Universal Robots PolyScope program: prac1_sergiorodriguez.urp

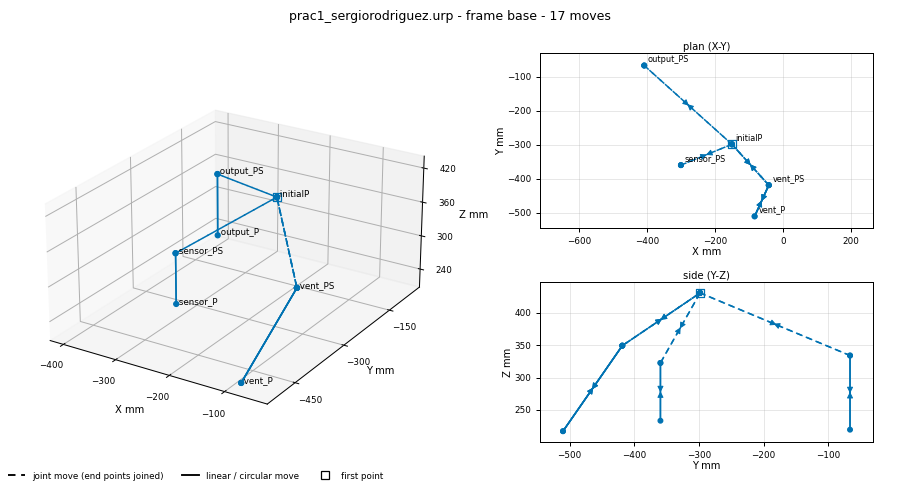
[picture p0: tool path of prac1_sergiorodriguez.urp in frame base, 17 of 17 moves have a stored position in this frame; points joined in program order, loops and branches not executed]
Program prac1_sergiorodriguez (installation=default directory=/programs createdIn=5.9.3.1031212 lastSavedIn=5.9.3.1031212 robotSerialNumber=20195300809)
Calibrated DH parameters: a=[-0.000085, -0.20076, -0.212369, 0.000121, -0.000118, 0]; d=[0.15185, -26.306375, 24.753047, 1.684739, 0.085386, 0.092088]; alpha=[1.572149, -0.00522, -0.011864, 1.571339, -1.571085, 0]; deltaTheta=[0, 0.599885, -0.513355, -0.086555, 0.000006, 0]
Robot Program (runOnlyOnce=false)
  URCap Gripper Activate (Robotiq_Grippers, Robotiq Inc.) dataModel(ResetAndActivateKey=false)
  URCap Gripper (Robotiq_Grippers, Robotiq Inc.) dataModel(position=0.0, force=100.0, speed=100.0, positionInDouble=0.0, forceInDouble=100.0, speedInDouble=100.0, slaveIds=[9], blocking=true)
  MoveJ speed 60 deg/s, acceleration 80 deg/s^2 (useActiveTCP=true) feature=Base
    Waypoint initialP: TCP in base x=-150.366 y=-298.238 z=430.772 mm, rx=1.2434 ry=2.8802 rz=0.0051 rad; joints [39.84, -76.565, 37.853, 308.981, -90.564, -2.908] deg
  Wait DigitalInput pin=digital_in[0]; digitalValue=1
  Wait Sleep waitTime=2.5
  MoveJ speed 60 deg/s, acceleration 80 deg/s^2 (useActiveTCP=true) feature=Base
    Waypoint sensor_PS: TCP in base x=-300.616 y=-359.588 z=322.64 mm, rx=0.0335 ry=-3.1211 rz=-0.1077 rad; joints [34.606, -41.931, 13.866, 299.406, -94.705, -56.283] deg
  MoveL speed 250 mm/s, acceleration 1200 mm/s^2 (useActiveTCP=true) feature=Base
    Waypoint sensor_P: TCP in base x=-300.596 y=-359.606 z=233.321 mm, rx=0.0335 ry=-3.1212 rz=-0.1078 rad; joints [34.589, -50.248, 53.908, 267.662, -94.751, -56.627] deg
  URCap Gripper (Robotiq_Grippers, Robotiq Inc.) dataModel(position=100.0, force=100.0, speed=100.0, positionInDouble=100.0, forceInDouble=100.0, speedInDouble=100.0, slaveIds=[9], blocking=true)
  Wait Sleep waitTime=1
  MoveL speed 250 mm/s, acceleration 1200 mm/s^2 (useActiveTCP=true) feature=Base
    Waypoint sensor_PS: TCP in base x=-300.616 y=-359.588 z=322.64 mm, rx=0.0335 ry=-3.1211 rz=-0.1077 rad; joints [34.606, -41.931, 13.866, 299.406, -94.705, -56.283] deg
  MoveJ speed 60 deg/s, acceleration 80 deg/s^2 (useActiveTCP=true) feature=Base
    Waypoint initialP: motionParameters(blendRadius=0.05); TCP in base x=-150.366 y=-298.238 z=430.772 mm, rx=1.2434 ry=2.8802 rz=0.0051 rad; joints [39.84, -76.565, 37.853, 308.981, -90.564, -2.908] deg
    Waypoint vent_PS: TCP in base x=-41.908 y=-418.605 z=349.288 mm, rx=0.042 ry=-3.1166 rz=0.0582 rad; joints [66.082, -63.586, 45.552, 285.498, -91.224, -25.238] deg
  MoveL speed 250 mm/s, acceleration 1200 mm/s^2 (useActiveTCP=true) feature=Base
    Waypoint vent_P: TCP in base x=-83.605 y=-510.387 z=217.125 mm, rx=-0.0383 ry=3.1266 rz=0.0695 rad; joints [66.078, -30.7, 21.233, 282.101, -91.231, -25.275] deg
    URCap Gripper (Robotiq_Grippers, Robotiq Inc.) dataModel(position=0.0, force=100.0, speed=100.0, positionInDouble=0.0, forceInDouble=100.0, speedInDouble=100.0, slaveIds=[9], blocking=true)
    Set DigitalOutput pin=digital_out[0]; digitalValue=0
    Waypoint vent_PS: TCP in base x=-41.908 y=-418.605 z=349.288 mm, rx=0.042 ry=-3.1166 rz=0.0582 rad; joints [66.082, -63.586, 45.552, 285.498, -91.224, -25.238] deg
  MoveJ speed 60 deg/s, acceleration 80 deg/s^2 (useActiveTCP=true) feature=Base
    Waypoint initialP: TCP in base x=-150.366 y=-298.238 z=430.772 mm, rx=1.2434 ry=2.8802 rz=0.0051 rad; joints [39.84, -76.565, 37.853, 308.981, -90.564, -2.908] deg
  Wait Sleep waitTime=5
  MoveJ speed 60 deg/s, acceleration 80 deg/s^2 (useActiveTCP=true) feature=Base
    Waypoint vent_PS: TCP in base x=-41.908 y=-418.605 z=349.288 mm, rx=0.042 ry=-3.1166 rz=0.0582 rad; joints [66.082, -63.586, 45.552, 285.498, -91.224, -25.238] deg
  MoveL speed 250 mm/s, acceleration 1200 mm/s^2 (useActiveTCP=true) feature=Base
    Waypoint vent_P: TCP in base x=-83.605 y=-510.387 z=217.125 mm, rx=-0.0383 ry=3.1266 rz=0.0695 rad; joints [66.078, -30.7, 21.233, 282.101, -91.231, -25.275] deg
    URCap Gripper (Robotiq_Grippers, Robotiq Inc.) dataModel(position=100.0, force=100.0, speed=100.0, positionInDouble=100.0, forceInDouble=100.0, speedInDouble=100.0, slaveIds=[9], blocking=true)
    Set DigitalOutput pin=digital_out[0]; digitalValue=0
    Wait Sleep waitTime=1
    Waypoint vent_PS: TCP in base x=-41.908 y=-418.605 z=349.288 mm, rx=0.042 ry=-3.1166 rz=0.0582 rad; joints [66.082, -63.586, 45.552, 285.498, -91.224, -25.238] deg
  MoveJ speed 60 deg/s, acceleration 80 deg/s^2 (useActiveTCP=true) feature=Base
    Waypoint initialP: motionParameters(blendRadius=0.05); TCP in base x=-150.366 y=-298.238 z=430.772 mm, rx=1.2434 ry=2.8802 rz=0.0051 rad; joints [39.84, -76.565, 37.853, 308.981, -90.564, -2.908] deg
    Waypoint output_PS: TCP in base x=-408.606 y=-66.295 z=334.079 mm, rx=-2.1876 ry=-2.2346 rz=0.059 rad; joints [-9.701, -66.872, 54.442, 280.524, -89.534, -10.707] deg
  MoveL speed 250 mm/s, acceleration 1200 mm/s^2 (useActiveTCP=true) feature=Base
    Waypoint output_P: TCP in base x=-408.608 y=-66.314 z=219.459 mm, rx=-2.1874 ry=-2.2345 rz=0.0591 rad; joints [-9.665, -65.617, 83.792, 249.915, -89.479, -11.032] deg
    URCap Gripper (Robotiq_Grippers, Robotiq Inc.) dataModel(position=0.0, force=100.0, speed=100.0, positionInDouble=0.0, forceInDouble=100.0, speedInDouble=100.0, slaveIds=[9], blocking=true)
    Wait Sleep waitTime=1
    Waypoint output_PS: TCP in base x=-408.606 y=-66.295 z=334.079 mm, rx=-2.1876 ry=-2.2346 rz=0.059 rad; joints [-9.701, -66.872, 54.442, 280.524, -89.534, -10.707] deg
  MoveJ speed 60 deg/s, acceleration 80 deg/s^2 (useActiveTCP=true) feature=Base
    Waypoint initialP: TCP in base x=-150.366 y=-298.238 z=430.772 mm, rx=1.2434 ry=2.8802 rz=0.0051 rad; joints [39.84, -76.565, 37.853, 308.981, -90.564, -2.908] deg
